// TIA Portal V20 export
FUNCTION_BLOCK "Main_Safety_RTG1"   // FB1, F_LAD
{ S7_Optimized_Access := 'TRUE' }
   VAR
      ESTOP1 : ESTOP1;
   END_VAR
BEGIN

REGION Network 1: Estops on electrical cabins
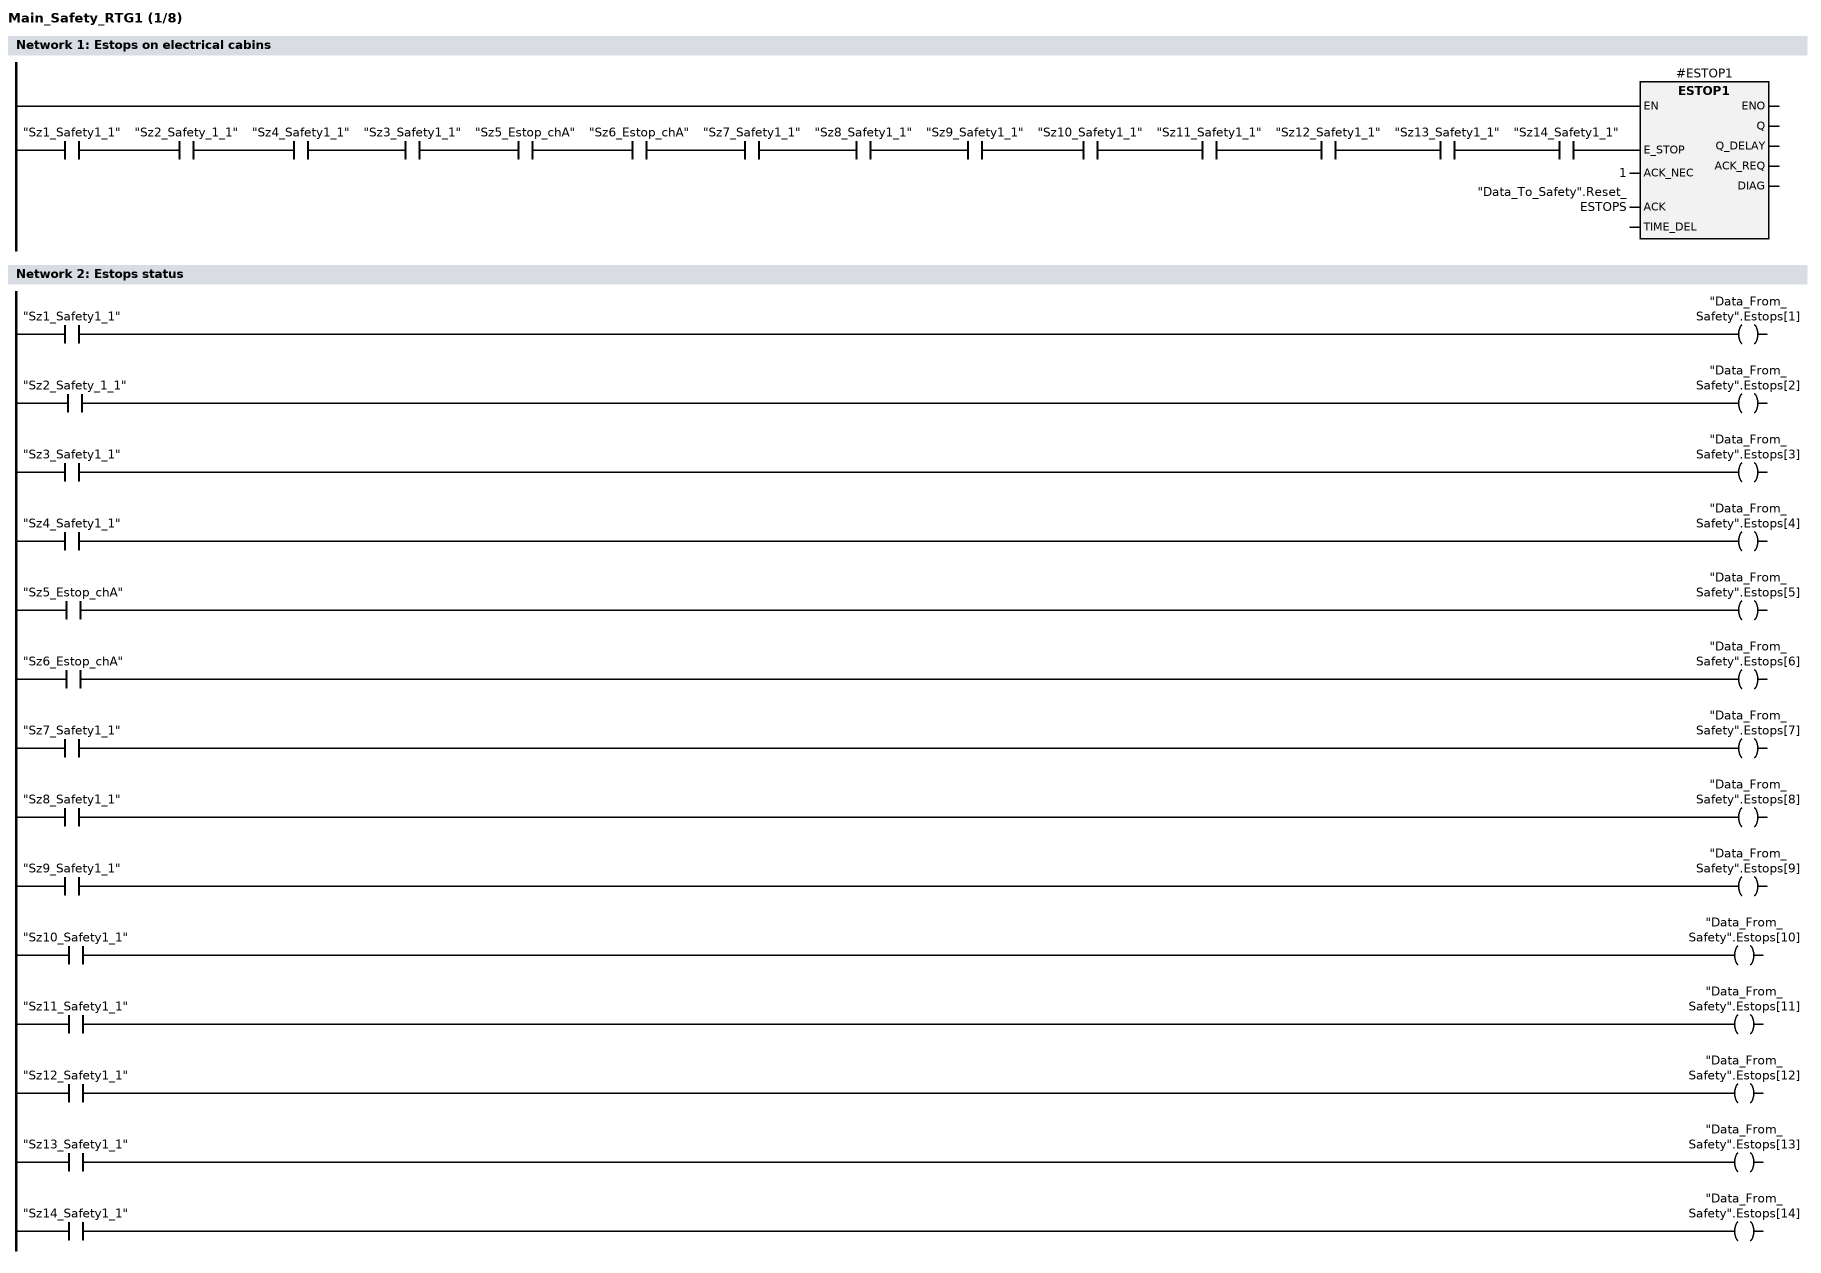
   RUNG wire#powerrail
      #ESTOP1.ESTOP1(E_STOP := wire#w1, ACK_NEC := 1, ACK := "Data_To_Safety".Reset_ESTOPS, TIME_DEL :=, Q =>, Q_DELAY =>, ACK_REQ =>, DIAG =>)
   END_RUNG
   RUNG wire#powerrail
      Contact( "Sz1_Safety1_1" )
      Contact( "Sz2_Safety_1_1" )
      Contact( "Sz4_Safety1_1" )
      Contact( "Sz3_Safety1_1" )
      Contact( "Sz5_Estop_chA" )
      Contact( "Sz6_Estop_chA" )
      Contact( "Sz7_Safety1_1" )
      Contact( "Sz8_Safety1_1" )
      Contact( "Sz9_Safety1_1" )
      Contact( "Sz10_Safety1_1" )
      Contact( "Sz11_Safety1_1" )
      Contact( "Sz12_Safety1_1" )
      Contact( "Sz13_Safety1_1" )
      Contact( "Sz14_Safety1_1" )
   END_RUNG wire#w1
   // the same network as SCL:
   #ESTOP1(E_STOP := "Sz1_Safety1_1" AND "Sz2_Safety_1_1" AND "Sz4_Safety1_1" AND "Sz3_Safety1_1" AND "Sz5_Estop_chA" AND "Sz6_Estop_chA" AND "Sz7_Safety1_1" AND "Sz8_Safety1_1" AND "Sz9_Safety1_1" AND "Sz10_Safety1_1" AND "Sz11_Safety1_1" AND "Sz12_Safety1_1" AND "Sz13_Safety1_1" AND "Sz14_Safety1_1",   // ESTOP1
           ACK_NEC := 1,
           ACK := "Data_To_Safety".Reset_ESTOPS);
END_REGION

REGION Network 2: Estops status
   RUNG wire#powerrail
      Contact( "Sz1_Safety1_1" )
      Coil( "Data_From_Safety".Estops[1] )
   END_RUNG
   RUNG wire#powerrail
      Contact( "Sz2_Safety_1_1" )
      Coil( "Data_From_Safety".Estops[2] )
   END_RUNG
   RUNG wire#powerrail
      Contact( "Sz3_Safety1_1" )
      Coil( "Data_From_Safety".Estops[3] )
   END_RUNG
   RUNG wire#powerrail
      Contact( "Sz4_Safety1_1" )
      Coil( "Data_From_Safety".Estops[4] )
   END_RUNG
   RUNG wire#powerrail
      Contact( "Sz5_Estop_chA" )
      Coil( "Data_From_Safety".Estops[5] )
   END_RUNG
   RUNG wire#powerrail
      Contact( "Sz6_Estop_chA" )
      Coil( "Data_From_Safety".Estops[6] )
   END_RUNG
   RUNG wire#powerrail
      Contact( "Sz7_Safety1_1" )
      Coil( "Data_From_Safety".Estops[7] )
   END_RUNG
   RUNG wire#powerrail
      Contact( "Sz8_Safety1_1" )
      Coil( "Data_From_Safety".Estops[8] )
   END_RUNG
   RUNG wire#powerrail
      Contact( "Sz9_Safety1_1" )
      Coil( "Data_From_Safety".Estops[9] )
   END_RUNG
   RUNG wire#powerrail
      Contact( "Sz10_Safety1_1" )
      Coil( "Data_From_Safety".Estops[10] )
   END_RUNG
   RUNG wire#powerrail
      Contact( "Sz11_Safety1_1" )
      Coil( "Data_From_Safety".Estops[11] )
   END_RUNG
   RUNG wire#powerrail
      Contact( "Sz12_Safety1_1" )
      Coil( "Data_From_Safety".Estops[12] )
   END_RUNG
   RUNG wire#powerrail
      Contact( "Sz13_Safety1_1" )
      Coil( "Data_From_Safety".Estops[13] )
   END_RUNG
   RUNG wire#powerrail
      Contact( "Sz14_Safety1_1" )
      Coil( "Data_From_Safety".Estops[14] )
   END_RUNG
   // the same network as SCL:
   "Data_From_Safety".Estops[1] := "Sz1_Safety1_1";
   "Data_From_Safety".Estops[2] := "Sz2_Safety_1_1";
   "Data_From_Safety".Estops[3] := "Sz3_Safety1_1";
   "Data_From_Safety".Estops[4] := "Sz4_Safety1_1";
   "Data_From_Safety".Estops[5] := "Sz5_Estop_chA";
   "Data_From_Safety".Estops[6] := "Sz6_Estop_chA";
   "Data_From_Safety".Estops[7] := "Sz7_Safety1_1";
   "Data_From_Safety".Estops[8] := "Sz8_Safety1_1";
   "Data_From_Safety".Estops[9] := "Sz9_Safety1_1";
   "Data_From_Safety".Estops[10] := "Sz10_Safety1_1";
   "Data_From_Safety".Estops[11] := "Sz11_Safety1_1";
   "Data_From_Safety".Estops[12] := "Sz12_Safety1_1";
   "Data_From_Safety".Estops[13] := "Sz13_Safety1_1";
   "Data_From_Safety".Estops[14] := "Sz14_Safety1_1";
END_REGION

REGION Network 3: Bumpers SS1_R1
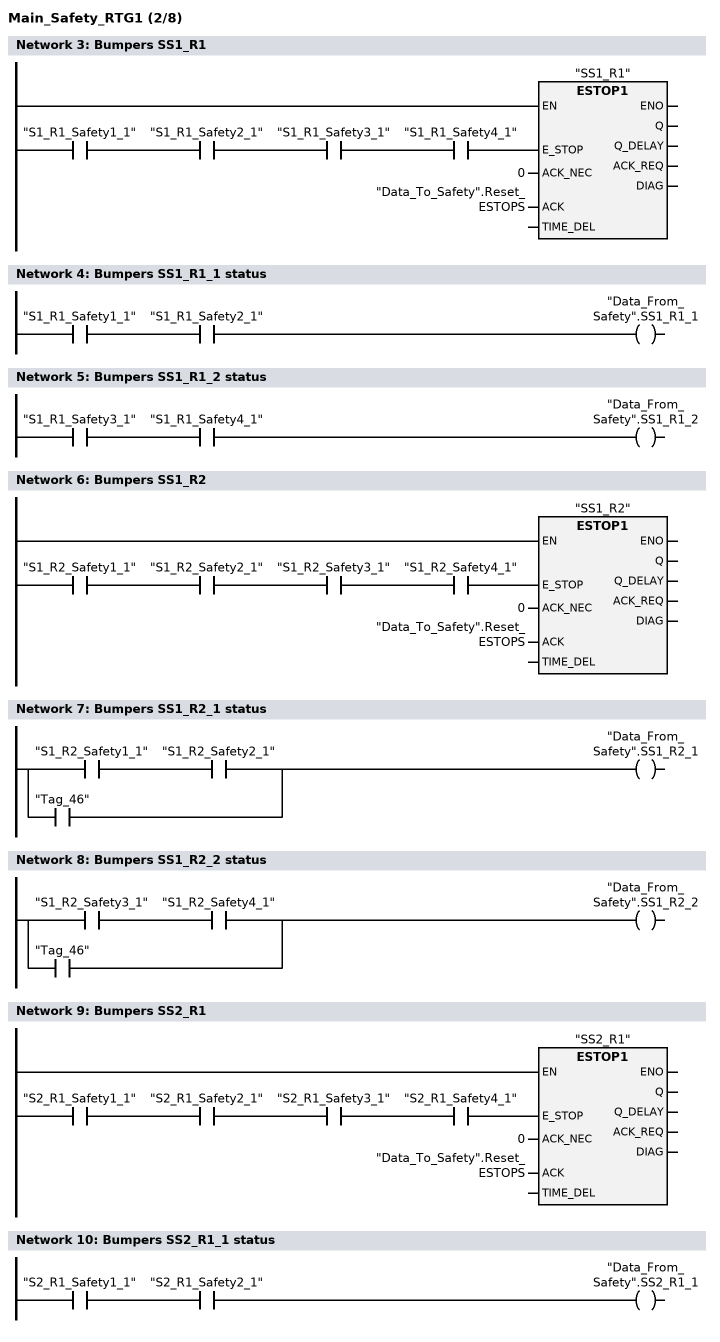
   RUNG wire#powerrail
      "SS1_R1".ESTOP1(E_STOP := wire#w1, ACK_NEC := 0, ACK := "Data_To_Safety".Reset_ESTOPS, TIME_DEL :=, Q =>, Q_DELAY =>, ACK_REQ =>, DIAG =>)
   END_RUNG
   RUNG wire#powerrail
      Contact( "S1_R1_Safety1_1" )
      Contact( "S1_R1_Safety2_1" )
      Contact( "S1_R1_Safety3_1" )
      Contact( "S1_R1_Safety4_1" )
   END_RUNG wire#w1
   // the same network as SCL:
   "SS1_R1"(E_STOP := "S1_R1_Safety1_1" AND "S1_R1_Safety2_1" AND "S1_R1_Safety3_1" AND "S1_R1_Safety4_1",   // ESTOP1
            ACK_NEC := 0,
            ACK := "Data_To_Safety".Reset_ESTOPS);
END_REGION

REGION Network 4: Bumpers SS1_R1_1 status
   RUNG wire#powerrail
      Contact( "S1_R1_Safety1_1" )
      Contact( "S1_R1_Safety2_1" )
      Coil( "Data_From_Safety".SS1_R1_1 )
   END_RUNG
   // the same network as SCL:
   "Data_From_Safety".SS1_R1_1 := "S1_R1_Safety1_1" AND "S1_R1_Safety2_1";
END_REGION

REGION Network 5: Bumpers SS1_R1_2 status
   RUNG wire#powerrail
      Contact( "S1_R1_Safety3_1" )
      Contact( "S1_R1_Safety4_1" )
      Coil( "Data_From_Safety".SS1_R1_2 )
   END_RUNG
   // the same network as SCL:
   "Data_From_Safety".SS1_R1_2 := "S1_R1_Safety3_1" AND "S1_R1_Safety4_1";
END_REGION

REGION Network 6: Bumpers SS1_R2
   RUNG wire#powerrail
      "SS1_R2".ESTOP1(E_STOP := wire#w1, ACK_NEC := 0, ACK := "Data_To_Safety".Reset_ESTOPS, TIME_DEL :=, Q =>, Q_DELAY =>, ACK_REQ =>, DIAG =>)
   END_RUNG
   RUNG wire#powerrail
      Contact( "S1_R2_Safety1_1" )
      Contact( "S1_R2_Safety2_1" )
      Contact( "S1_R2_Safety3_1" )
      Contact( "S1_R2_Safety4_1" )
   END_RUNG wire#w1
   // the same network as SCL:
   "SS1_R2"(E_STOP := "S1_R2_Safety1_1" AND "S1_R2_Safety2_1" AND "S1_R2_Safety3_1" AND "S1_R2_Safety4_1",   // ESTOP1
            ACK_NEC := 0,
            ACK := "Data_To_Safety".Reset_ESTOPS);
END_REGION

REGION Network 7: Bumpers SS1_R2_1 status
   RUNG wire#powerrail
      Contact( "S1_R2_Safety1_1" )
      Contact( "S1_R2_Safety2_1" )
      wire#w1
      Coil( "Data_From_Safety".SS1_R2_1 )
   END_RUNG
   RUNG wire#powerrail
      Contact( "Tag_46" )
   END_RUNG wire#w1
   // the same network as SCL:
   "Data_From_Safety".SS1_R2_1 := ("S1_R2_Safety1_1" AND "S1_R2_Safety2_1") OR "Tag_46";
END_REGION

REGION Network 8: Bumpers SS1_R2_2 status
   RUNG wire#powerrail
      Contact( "S1_R2_Safety3_1" )
      Contact( "S1_R2_Safety4_1" )
      wire#w1
      Coil( "Data_From_Safety".SS1_R2_2 )
   END_RUNG
   RUNG wire#powerrail
      Contact( "Tag_46" )
   END_RUNG wire#w1
   // the same network as SCL:
   "Data_From_Safety".SS1_R2_2 := ("S1_R2_Safety3_1" AND "S1_R2_Safety4_1") OR "Tag_46";
END_REGION

REGION Network 9: Bumpers SS2_R1
   RUNG wire#powerrail
      "SS2_R1".ESTOP1(E_STOP := wire#w1, ACK_NEC := 0, ACK := "Data_To_Safety".Reset_ESTOPS, TIME_DEL :=, Q =>, Q_DELAY =>, ACK_REQ =>, DIAG =>)
   END_RUNG
   RUNG wire#powerrail
      Contact( "S2_R1_Safety1_1" )
      Contact( "S2_R1_Safety2_1" )
      Contact( "S2_R1_Safety3_1" )
      Contact( "S2_R1_Safety4_1" )
   END_RUNG wire#w1
   // the same network as SCL:
   "SS2_R1"(E_STOP := "S2_R1_Safety1_1" AND "S2_R1_Safety2_1" AND "S2_R1_Safety3_1" AND "S2_R1_Safety4_1",   // ESTOP1
            ACK_NEC := 0,
            ACK := "Data_To_Safety".Reset_ESTOPS);
END_REGION

REGION Network 10: Bumpers SS2_R1_1 status
   RUNG wire#powerrail
      Contact( "S2_R1_Safety1_1" )
      Contact( "S2_R1_Safety2_1" )
      Coil( "Data_From_Safety".SS2_R1_1 )
   END_RUNG
   // the same network as SCL:
   "Data_From_Safety".SS2_R1_1 := "S2_R1_Safety1_1" AND "S2_R1_Safety2_1";
END_REGION

REGION Network 11: Bumpers SS2_R1_2 status
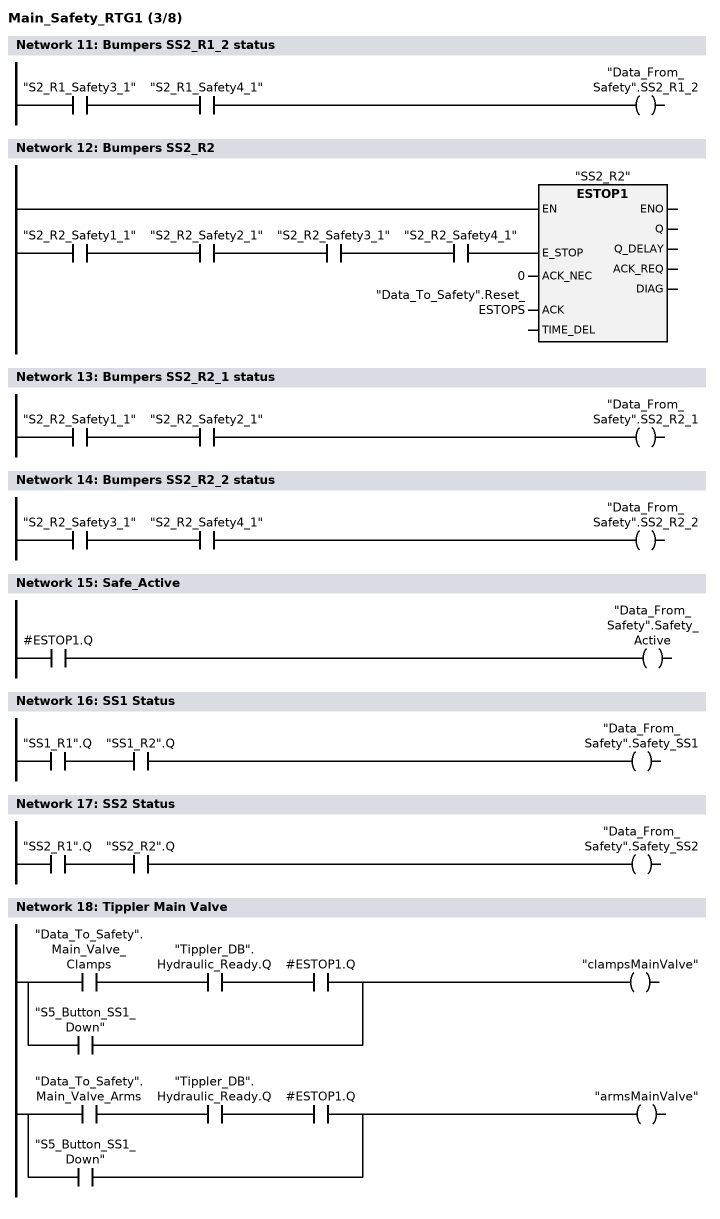
   RUNG wire#powerrail
      Contact( "S2_R1_Safety3_1" )
      Contact( "S2_R1_Safety4_1" )
      Coil( "Data_From_Safety".SS2_R1_2 )
   END_RUNG
   // the same network as SCL:
   "Data_From_Safety".SS2_R1_2 := "S2_R1_Safety3_1" AND "S2_R1_Safety4_1";
END_REGION

REGION Network 12: Bumpers SS2_R2
   RUNG wire#powerrail
      "SS2_R2".ESTOP1(E_STOP := wire#w1, ACK_NEC := 0, ACK := "Data_To_Safety".Reset_ESTOPS, TIME_DEL :=, Q =>, Q_DELAY =>, ACK_REQ =>, DIAG =>)
   END_RUNG
   RUNG wire#powerrail
      Contact( "S2_R2_Safety1_1" )
      Contact( "S2_R2_Safety2_1" )
      Contact( "S2_R2_Safety3_1" )
      Contact( "S2_R2_Safety4_1" )
   END_RUNG wire#w1
   // the same network as SCL:
   "SS2_R2"(E_STOP := "S2_R2_Safety1_1" AND "S2_R2_Safety2_1" AND "S2_R2_Safety3_1" AND "S2_R2_Safety4_1",   // ESTOP1
            ACK_NEC := 0,
            ACK := "Data_To_Safety".Reset_ESTOPS);
END_REGION

REGION Network 13: Bumpers SS2_R2_1 status
   RUNG wire#powerrail
      Contact( "S2_R2_Safety1_1" )
      Contact( "S2_R2_Safety2_1" )
      Coil( "Data_From_Safety".SS2_R2_1 )
   END_RUNG
   // the same network as SCL:
   "Data_From_Safety".SS2_R2_1 := "S2_R2_Safety1_1" AND "S2_R2_Safety2_1";
END_REGION

REGION Network 14: Bumpers SS2_R2_2 status
   RUNG wire#powerrail
      Contact( "S2_R2_Safety3_1" )
      Contact( "S2_R2_Safety4_1" )
      Coil( "Data_From_Safety".SS2_R2_2 )
   END_RUNG
   // the same network as SCL:
   "Data_From_Safety".SS2_R2_2 := "S2_R2_Safety3_1" AND "S2_R2_Safety4_1";
END_REGION

REGION Network 15: Safe_Active
   RUNG wire#powerrail
      Contact( #ESTOP1.Q )
      Coil( "Data_From_Safety".Safety_Active )
   END_RUNG
   // the same network as SCL:
   "Data_From_Safety".Safety_Active := #ESTOP1.Q;
END_REGION

REGION Network 16: SS1 Status
   RUNG wire#powerrail
      Contact( "SS1_R1".Q )
      Contact( "SS1_R2".Q )
      Coil( "Data_From_Safety".Safety_SS1 )
   END_RUNG
   // the same network as SCL:
   "Data_From_Safety".Safety_SS1 := "SS1_R1".Q AND "SS1_R2".Q;
END_REGION

REGION Network 17: SS2 Status
   RUNG wire#powerrail
      Contact( "SS2_R1".Q )
      Contact( "SS2_R2".Q )
      Coil( "Data_From_Safety".Safety_SS2 )
   END_RUNG
   // the same network as SCL:
   "Data_From_Safety".Safety_SS2 := "SS2_R1".Q AND "SS2_R2".Q;
END_REGION

REGION Network 18: Tippler Main Valve
   RUNG wire#powerrail
      Contact( "Data_To_Safety".Main_Valve_Clamps )
      Contact( "Tippler_DB".Hydraulic_Ready.Q )
      Contact( #ESTOP1.Q )
      wire#w1
      Coil( "clampsMainValve" )
   END_RUNG
   RUNG wire#powerrail
      Contact( "S5_Button_SS1_Down" )
   END_RUNG wire#w1
   RUNG wire#powerrail
      Contact( "Data_To_Safety".Main_Valve_Arms )
      Contact( "Tippler_DB".Hydraulic_Ready.Q )
      Contact( #ESTOP1.Q )
      wire#w2
      Coil( "armsMainValve" )
   END_RUNG
   RUNG wire#powerrail
      Contact( "S5_Button_SS1_Down" )
   END_RUNG wire#w2
   // the same network as SCL:
   "clampsMainValve" := ("Data_To_Safety".Main_Valve_Clamps AND "Tippler_DB".Hydraulic_Ready.Q AND #ESTOP1.Q) OR "S5_Button_SS1_Down";
   "armsMainValve" := ("Data_To_Safety".Main_Valve_Arms AND "Tippler_DB".Hydraulic_Ready.Q AND #ESTOP1.Q) OR "S5_Button_SS1_Down";
END_REGION

REGION Network 19: S0_R1, S0_R2
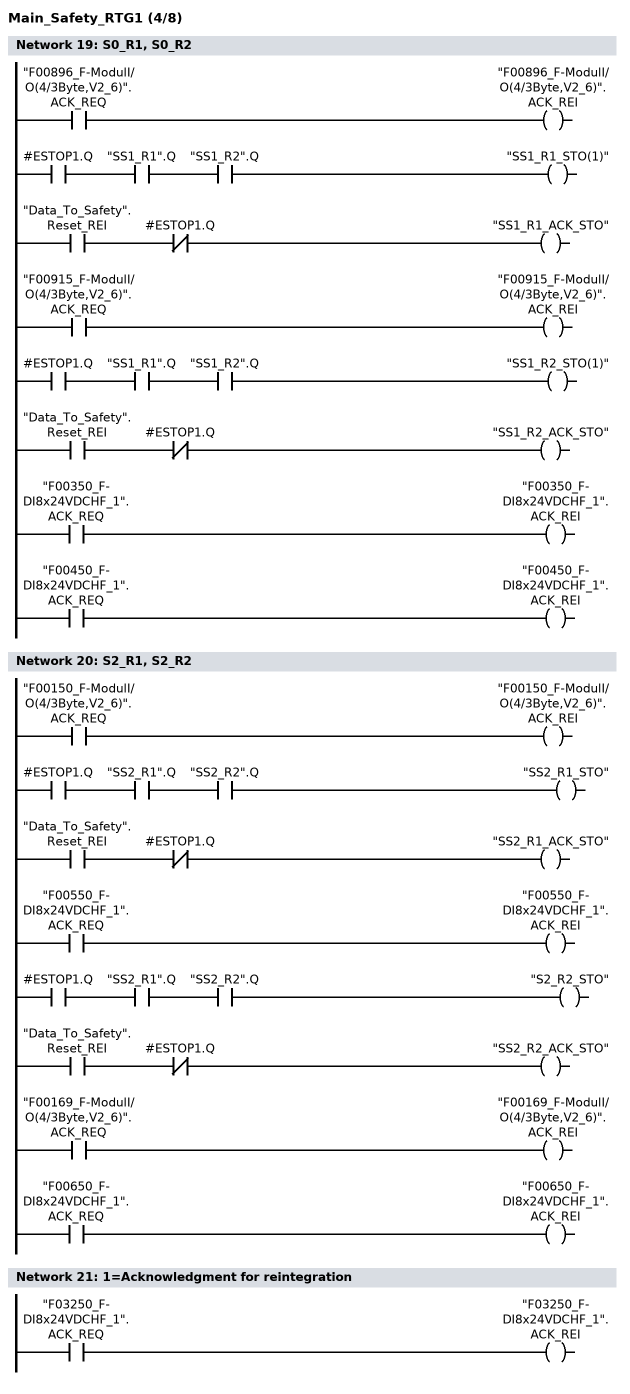
   RUNG wire#powerrail
      Contact( "F00896_F-ModulI/O(4/3Byte,V2_6)".ACK_REQ )
      Coil( "F00896_F-ModulI/O(4/3Byte,V2_6)".ACK_REI )
   END_RUNG
   RUNG wire#powerrail
      Contact( #ESTOP1.Q )
      Contact( "SS1_R1".Q )
      Contact( "SS1_R2".Q )
      Coil( "SS1_R1_STO(1)" )
   END_RUNG
   RUNG wire#powerrail
      Contact( "Data_To_Safety".Reset_REI )
      I_Contact( #ESTOP1.Q )
      Coil( "SS1_R1_ACK_STO" )
   END_RUNG
   RUNG wire#powerrail
      Contact( "F00915_F-ModulI/O(4/3Byte,V2_6)".ACK_REQ )
      Coil( "F00915_F-ModulI/O(4/3Byte,V2_6)".ACK_REI )
   END_RUNG
   RUNG wire#powerrail
      Contact( #ESTOP1.Q )
      Contact( "SS1_R1".Q )
      Contact( "SS1_R2".Q )
      Coil( "SS1_R2_STO(1)" )
   END_RUNG
   RUNG wire#powerrail
      Contact( "Data_To_Safety".Reset_REI )
      I_Contact( #ESTOP1.Q )
      Coil( "SS1_R2_ACK_STO" )
   END_RUNG
   RUNG wire#powerrail
      Contact( "F00350_F-DI8x24VDCHF_1".ACK_REQ )
      Coil( "F00350_F-DI8x24VDCHF_1".ACK_REI )
   END_RUNG
   RUNG wire#powerrail
      Contact( "F00450_F-DI8x24VDCHF_1".ACK_REQ )
      Coil( "F00450_F-DI8x24VDCHF_1".ACK_REI )
   END_RUNG
   // the same network as SCL:
   "F00896_F-ModulI/O(4/3Byte,V2_6)".ACK_REI := "F00896_F-ModulI/O(4/3Byte,V2_6)".ACK_REQ;
   "SS1_R1_STO(1)" := #ESTOP1.Q AND "SS1_R1".Q AND "SS1_R2".Q;
   "SS1_R1_ACK_STO" := "Data_To_Safety".Reset_REI AND NOT #ESTOP1.Q;
   "F00915_F-ModulI/O(4/3Byte,V2_6)".ACK_REI := "F00915_F-ModulI/O(4/3Byte,V2_6)".ACK_REQ;
   "SS1_R2_STO(1)" := #ESTOP1.Q AND "SS1_R1".Q AND "SS1_R2".Q;
   "SS1_R2_ACK_STO" := "Data_To_Safety".Reset_REI AND NOT #ESTOP1.Q;
   "F00350_F-DI8x24VDCHF_1".ACK_REI := "F00350_F-DI8x24VDCHF_1".ACK_REQ;
   "F00450_F-DI8x24VDCHF_1".ACK_REI := "F00450_F-DI8x24VDCHF_1".ACK_REQ;
END_REGION

REGION Network 20: S2_R1, S2_R2
   RUNG wire#powerrail
      Contact( "F00150_F-ModulI/O(4/3Byte,V2_6)".ACK_REQ )
      Coil( "F00150_F-ModulI/O(4/3Byte,V2_6)".ACK_REI )
   END_RUNG
   RUNG wire#powerrail
      Contact( #ESTOP1.Q )
      Contact( "SS2_R1".Q )
      Contact( "SS2_R2".Q )
      Coil( "SS2_R1_STO" )
   END_RUNG
   RUNG wire#powerrail
      Contact( "Data_To_Safety".Reset_REI )
      I_Contact( #ESTOP1.Q )
      Coil( "SS2_R1_ACK_STO" )
   END_RUNG
   RUNG wire#powerrail
      Contact( "F00550_F-DI8x24VDCHF_1".ACK_REQ )
      Coil( "F00550_F-DI8x24VDCHF_1".ACK_REI )
   END_RUNG
   RUNG wire#powerrail
      Contact( #ESTOP1.Q )
      Contact( "SS2_R1".Q )
      Contact( "SS2_R2".Q )
      Coil( "S2_R2_STO" )
   END_RUNG
   RUNG wire#powerrail
      Contact( "Data_To_Safety".Reset_REI )
      I_Contact( #ESTOP1.Q )
      Coil( "SS2_R2_ACK_STO" )
   END_RUNG
   RUNG wire#powerrail
      Contact( "F00169_F-ModulI/O(4/3Byte,V2_6)".ACK_REQ )
      Coil( "F00169_F-ModulI/O(4/3Byte,V2_6)".ACK_REI )
   END_RUNG
   RUNG wire#powerrail
      Contact( "F00650_F-DI8x24VDCHF_1".ACK_REQ )
      Coil( "F00650_F-DI8x24VDCHF_1".ACK_REI )
   END_RUNG
   // the same network as SCL:
   "F00150_F-ModulI/O(4/3Byte,V2_6)".ACK_REI := "F00150_F-ModulI/O(4/3Byte,V2_6)".ACK_REQ;
   "SS2_R1_STO" := #ESTOP1.Q AND "SS2_R1".Q AND "SS2_R2".Q;
   "SS2_R1_ACK_STO" := "Data_To_Safety".Reset_REI AND NOT #ESTOP1.Q;
   "F00550_F-DI8x24VDCHF_1".ACK_REI := "F00550_F-DI8x24VDCHF_1".ACK_REQ;
   "S2_R2_STO" := #ESTOP1.Q AND "SS2_R1".Q AND "SS2_R2".Q;
   "SS2_R2_ACK_STO" := "Data_To_Safety".Reset_REI AND NOT #ESTOP1.Q;
   "F00169_F-ModulI/O(4/3Byte,V2_6)".ACK_REI := "F00169_F-ModulI/O(4/3Byte,V2_6)".ACK_REQ;
   "F00650_F-DI8x24VDCHF_1".ACK_REI := "F00650_F-DI8x24VDCHF_1".ACK_REQ;
END_REGION

REGION Network 21: 1=Acknowledgment for reintegration
   RUNG wire#powerrail
      Contact( "F03250_F-DI8x24VDCHF_1".ACK_REQ )
      Coil( "F03250_F-DI8x24VDCHF_1".ACK_REI )
   END_RUNG
   // the same network as SCL:
   "F03250_F-DI8x24VDCHF_1".ACK_REI := "F03250_F-DI8x24VDCHF_1".ACK_REQ;
END_REGION

REGION Network 22: ROW 1
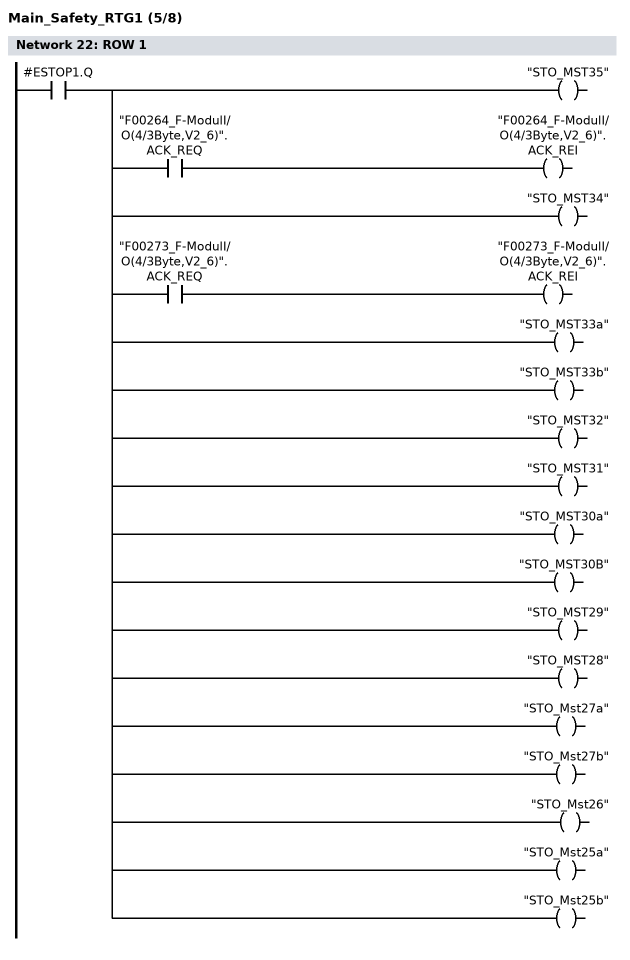
   RUNG wire#powerrail
      Contact( #ESTOP1.Q )
      wire#w1
      Coil( "STO_MST35" )
   END_RUNG
   RUNG wire#w1
      Contact( "F00264_F-ModulI/O(4/3Byte,V2_6)".ACK_REQ )
      Coil( "F00264_F-ModulI/O(4/3Byte,V2_6)".ACK_REI )
   END_RUNG
   RUNG wire#w1
      Coil( "STO_MST34" )
   END_RUNG
   RUNG wire#w1
      Contact( "F00273_F-ModulI/O(4/3Byte,V2_6)".ACK_REQ )
      Coil( "F00273_F-ModulI/O(4/3Byte,V2_6)".ACK_REI )
   END_RUNG
   RUNG wire#w1
      Coil( "STO_MST33a" )
   END_RUNG
   RUNG wire#w1
      Coil( "STO_MST33b" )
   END_RUNG
   RUNG wire#w1
      Coil( "STO_MST32" )
   END_RUNG
   RUNG wire#w1
      Coil( "STO_MST31" )
   END_RUNG
   RUNG wire#w1
      Coil( "STO_MST30a" )
   END_RUNG
   RUNG wire#w1
      Coil( "STO_MST30B" )
   END_RUNG
   RUNG wire#w1
      Coil( "STO_MST29" )
   END_RUNG
   RUNG wire#w1
      Coil( "STO_MST28" )
   END_RUNG
   RUNG wire#w1
      Coil( "STO_Mst27a" )
   END_RUNG
   RUNG wire#w1
      Coil( "STO_Mst27b" )
   END_RUNG
   RUNG wire#w1
      Coil( "STO_Mst26" )
   END_RUNG
   RUNG wire#w1
      Coil( "STO_Mst25a" )
   END_RUNG
   RUNG wire#w1
      Coil( "STO_Mst25b" )
   END_RUNG
   // the same network as SCL:
   "STO_MST35" := #ESTOP1.Q;
   "F00264_F-ModulI/O(4/3Byte,V2_6)".ACK_REI := #ESTOP1.Q AND "F00264_F-ModulI/O(4/3Byte,V2_6)".ACK_REQ;
   "STO_MST34" := #ESTOP1.Q;
   "F00273_F-ModulI/O(4/3Byte,V2_6)".ACK_REI := #ESTOP1.Q AND "F00273_F-ModulI/O(4/3Byte,V2_6)".ACK_REQ;
   "STO_MST33a" := #ESTOP1.Q;
   "STO_MST33b" := #ESTOP1.Q;
   "STO_MST32" := #ESTOP1.Q;
   "STO_MST31" := #ESTOP1.Q;
   "STO_MST30a" := #ESTOP1.Q;
   "STO_MST30B" := #ESTOP1.Q;
   "STO_MST29" := #ESTOP1.Q;
   "STO_MST28" := #ESTOP1.Q;
   "STO_Mst27a" := #ESTOP1.Q;
   "STO_Mst27b" := #ESTOP1.Q;
   "STO_Mst26" := #ESTOP1.Q;
   "STO_Mst25a" := #ESTOP1.Q;
   "STO_Mst25b" := #ESTOP1.Q;
END_REGION

REGION Network 23: ROW 2
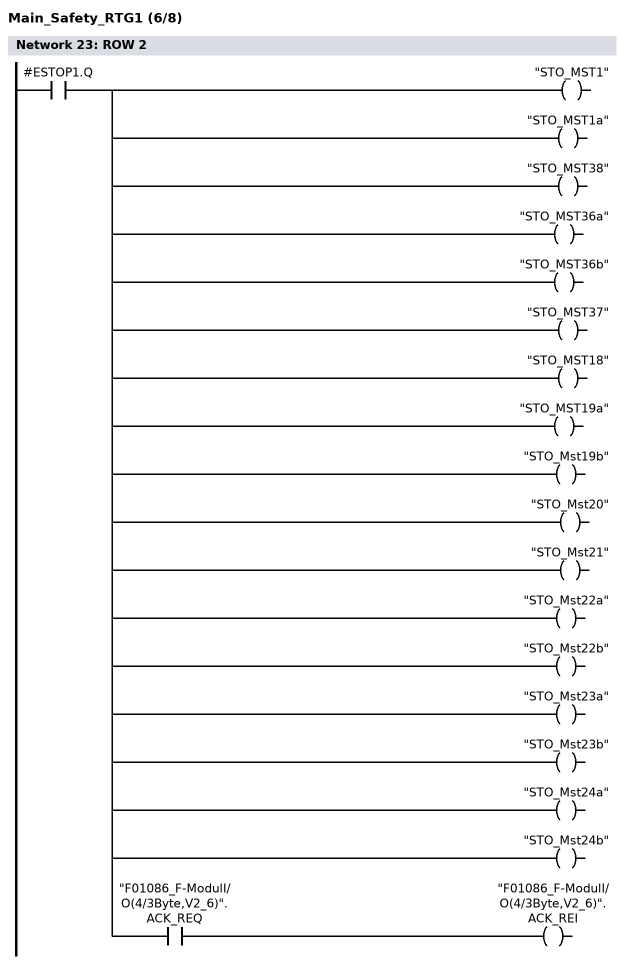
   RUNG wire#powerrail
      Contact( #ESTOP1.Q )
      wire#w1
      Coil( "STO_MST1" )
   END_RUNG
   RUNG wire#w1
      Coil( "STO_MST1a" )
   END_RUNG
   RUNG wire#w1
      Coil( "STO_MST38" )
   END_RUNG
   RUNG wire#w1
      Coil( "STO_MST36a" )
   END_RUNG
   RUNG wire#w1
      Coil( "STO_MST36b" )
   END_RUNG
   RUNG wire#w1
      Coil( "STO_MST37" )
   END_RUNG
   RUNG wire#w1
      Coil( "STO_MST18" )
   END_RUNG
   RUNG wire#w1
      Coil( "STO_MST19a" )
   END_RUNG
   RUNG wire#w1
      Coil( "STO_Mst19b" )
   END_RUNG
   RUNG wire#w1
      Coil( "STO_Mst20" )
   END_RUNG
   RUNG wire#w1
      Coil( "STO_Mst21" )
   END_RUNG
   RUNG wire#w1
      Coil( "STO_Mst22a" )
   END_RUNG
   RUNG wire#w1
      Coil( "STO_Mst22b" )
   END_RUNG
   RUNG wire#w1
      Coil( "STO_Mst23a" )
   END_RUNG
   RUNG wire#w1
      Coil( "STO_Mst23b" )
   END_RUNG
   RUNG wire#w1
      Coil( "STO_Mst24a" )
   END_RUNG
   RUNG wire#w1
      Coil( "STO_Mst24b" )
   END_RUNG
   RUNG wire#w1
      Contact( "F01086_F-ModulI/O(4/3Byte,V2_6)".ACK_REQ )
      Coil( "F01086_F-ModulI/O(4/3Byte,V2_6)".ACK_REI )
   END_RUNG
   // the same network as SCL:
   "STO_MST1" := #ESTOP1.Q;
   "STO_MST1a" := #ESTOP1.Q;
   "STO_MST38" := #ESTOP1.Q;
   "STO_MST36a" := #ESTOP1.Q;
   "STO_MST36b" := #ESTOP1.Q;
   "STO_MST37" := #ESTOP1.Q;
   "STO_MST18" := #ESTOP1.Q;
   "STO_MST19a" := #ESTOP1.Q;
   "STO_Mst19b" := #ESTOP1.Q;
   "STO_Mst20" := #ESTOP1.Q;
   "STO_Mst21" := #ESTOP1.Q;
   "STO_Mst22a" := #ESTOP1.Q;
   "STO_Mst22b" := #ESTOP1.Q;
   "STO_Mst23a" := #ESTOP1.Q;
   "STO_Mst23b" := #ESTOP1.Q;
   "STO_Mst24a" := #ESTOP1.Q;
   "STO_Mst24b" := #ESTOP1.Q;
   "F01086_F-ModulI/O(4/3Byte,V2_6)".ACK_REI := #ESTOP1.Q AND "F01086_F-ModulI/O(4/3Byte,V2_6)".ACK_REQ;
END_REGION

REGION Network 24: ROW 4
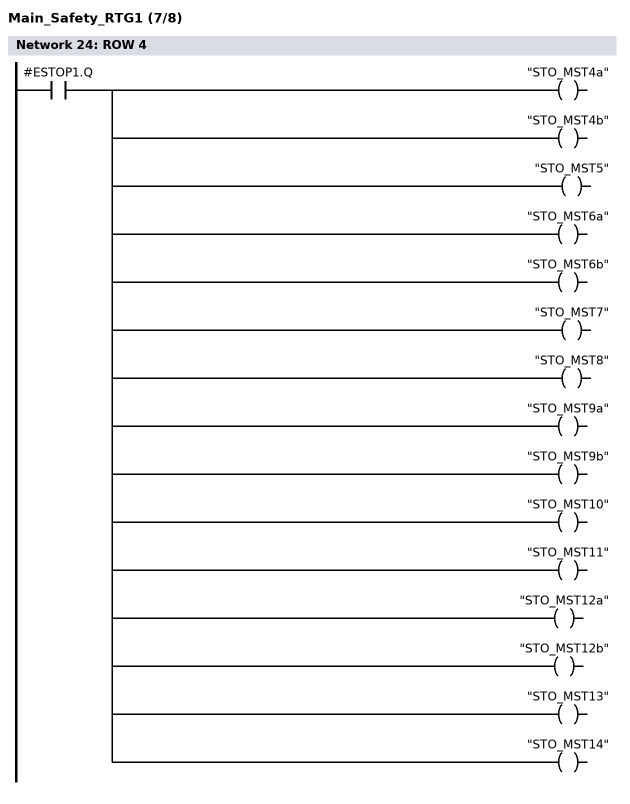
   RUNG wire#powerrail
      Contact( #ESTOP1.Q )
      wire#w1
      Coil( "STO_MST4a" )
   END_RUNG
   RUNG wire#w1
      Coil( "STO_MST4b" )
   END_RUNG
   RUNG wire#w1
      Coil( "STO_MST5" )
   END_RUNG
   RUNG wire#w1
      Coil( "STO_MST6a" )
   END_RUNG
   RUNG wire#w1
      Coil( "STO_MST6b" )
   END_RUNG
   RUNG wire#w1
      Coil( "STO_MST7" )
   END_RUNG
   RUNG wire#w1
      Coil( "STO_MST8" )
   END_RUNG
   RUNG wire#w1
      Coil( "STO_MST9a" )
   END_RUNG
   RUNG wire#w1
      Coil( "STO_MST9b" )
   END_RUNG
   RUNG wire#w1
      Coil( "STO_MST10" )
   END_RUNG
   RUNG wire#w1
      Coil( "STO_MST11" )
   END_RUNG
   RUNG wire#w1
      Coil( "STO_MST12a" )
   END_RUNG
   RUNG wire#w1
      Coil( "STO_MST12b" )
   END_RUNG
   RUNG wire#w1
      Coil( "STO_MST13" )
   END_RUNG
   RUNG wire#w1
      Coil( "STO_MST14" )
   END_RUNG
   // the same network as SCL:
   "STO_MST4a" := #ESTOP1.Q;
   "STO_MST4b" := #ESTOP1.Q;
   "STO_MST5" := #ESTOP1.Q;
   "STO_MST6a" := #ESTOP1.Q;
   "STO_MST6b" := #ESTOP1.Q;
   "STO_MST7" := #ESTOP1.Q;
   "STO_MST8" := #ESTOP1.Q;
   "STO_MST9a" := #ESTOP1.Q;
   "STO_MST9b" := #ESTOP1.Q;
   "STO_MST10" := #ESTOP1.Q;
   "STO_MST11" := #ESTOP1.Q;
   "STO_MST12a" := #ESTOP1.Q;
   "STO_MST12b" := #ESTOP1.Q;
   "STO_MST13" := #ESTOP1.Q;
   "STO_MST14" := #ESTOP1.Q;
END_REGION

REGION Network 25: CS
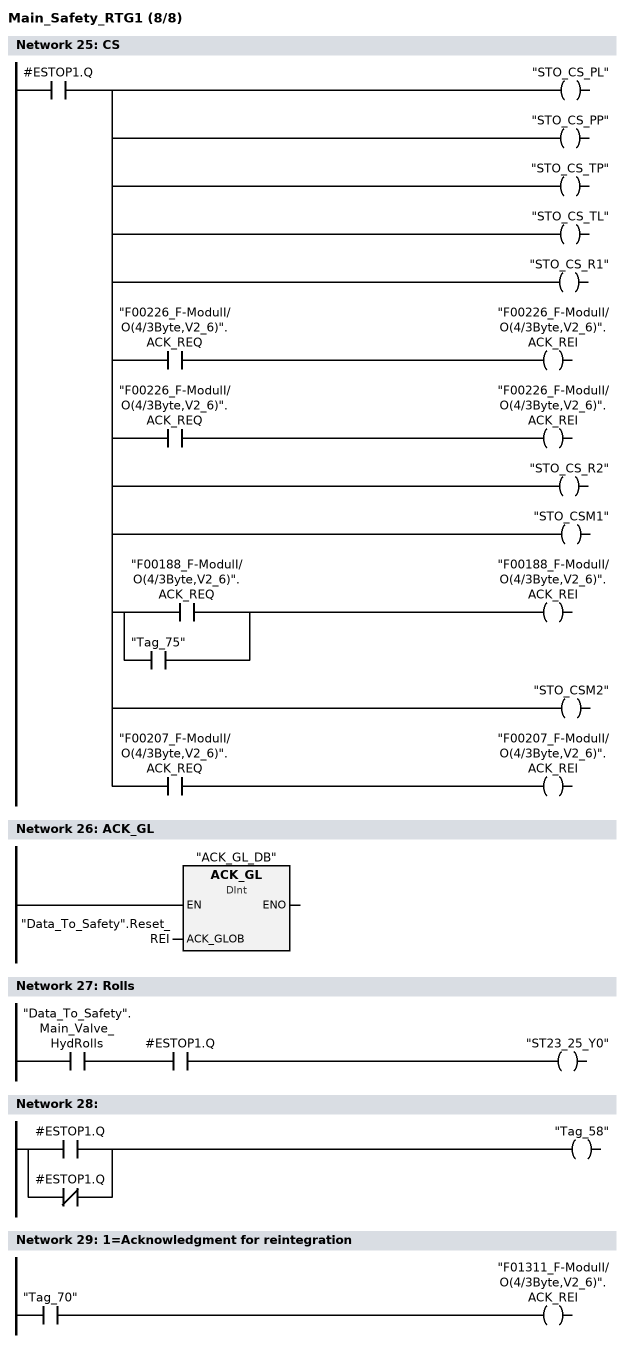
   RUNG wire#powerrail
      Contact( #ESTOP1.Q )
      wire#w1
      Coil( "STO_CS_PL" )
   END_RUNG
   RUNG wire#w1
      Coil( "STO_CS_PP" )
   END_RUNG
   RUNG wire#w1
      Coil( "STO_CS_TP" )
   END_RUNG
   RUNG wire#w1
      Coil( "STO_CS_TL" )
   END_RUNG
   RUNG wire#w1
      Coil( "STO_CS_R1" )
   END_RUNG
   RUNG wire#w1
      Contact( "F00226_F-ModulI/O(4/3Byte,V2_6)".ACK_REQ )
      Coil( "F00226_F-ModulI/O(4/3Byte,V2_6)".ACK_REI )
   END_RUNG
   RUNG wire#w1
      Contact( "F00226_F-ModulI/O(4/3Byte,V2_6)".ACK_REQ )
      Coil( "F00226_F-ModulI/O(4/3Byte,V2_6)".ACK_REI )
   END_RUNG
   RUNG wire#w1
      Coil( "STO_CS_R2" )
   END_RUNG
   RUNG wire#w1
      Coil( "STO_CSM1" )
   END_RUNG
   RUNG wire#w1
      Contact( "F00188_F-ModulI/O(4/3Byte,V2_6)".ACK_REQ )
      wire#w2
      Coil( "F00188_F-ModulI/O(4/3Byte,V2_6)".ACK_REI )
   END_RUNG
   RUNG wire#w1
      Contact( "Tag_75" )
   END_RUNG wire#w2
   RUNG wire#w1
      Coil( "STO_CSM2" )
   END_RUNG
   RUNG wire#w1
      Contact( "F00207_F-ModulI/O(4/3Byte,V2_6)".ACK_REQ )
      Coil( "F00207_F-ModulI/O(4/3Byte,V2_6)".ACK_REI )
   END_RUNG
   // the same network as SCL:
   "STO_CS_PL" := #ESTOP1.Q;
   "STO_CS_PP" := #ESTOP1.Q;
   "STO_CS_TP" := #ESTOP1.Q;
   "STO_CS_TL" := #ESTOP1.Q;
   "STO_CS_R1" := #ESTOP1.Q;
   "F00226_F-ModulI/O(4/3Byte,V2_6)".ACK_REI := #ESTOP1.Q AND "F00226_F-ModulI/O(4/3Byte,V2_6)".ACK_REQ;
   "F00226_F-ModulI/O(4/3Byte,V2_6)".ACK_REI := #ESTOP1.Q AND "F00226_F-ModulI/O(4/3Byte,V2_6)".ACK_REQ;
   "STO_CS_R2" := #ESTOP1.Q;
   "STO_CSM1" := #ESTOP1.Q;
   "F00188_F-ModulI/O(4/3Byte,V2_6)".ACK_REI := #ESTOP1.Q AND ("F00188_F-ModulI/O(4/3Byte,V2_6)".ACK_REQ OR "Tag_75");
   "STO_CSM2" := #ESTOP1.Q;
   "F00207_F-ModulI/O(4/3Byte,V2_6)".ACK_REI := #ESTOP1.Q AND "F00207_F-ModulI/O(4/3Byte,V2_6)".ACK_REQ;
END_REGION

REGION Network 26: ACK_GL
   RUNG wire#powerrail
      { S7_Templates := "codedbool_type := DInt" } "ACK_GL_DB".ACK_GL(ACK_GLOB := "Data_To_Safety".Reset_REI)
   END_RUNG
   // the same network as SCL:
   "ACK_GL_DB"(ACK_GLOB := "Data_To_Safety".Reset_REI);   // ACK_GL
END_REGION

REGION Network 27: Rolls
   RUNG wire#powerrail
      Contact( "Data_To_Safety".Main_Valve_HydRolls )
      Contact( #ESTOP1.Q )
      Coil( "ST23_25_Y0" )
   END_RUNG
   // the same network as SCL:
   "ST23_25_Y0" := "Data_To_Safety".Main_Valve_HydRolls AND #ESTOP1.Q;
END_REGION

REGION Network 28
   RUNG wire#powerrail
      Contact( #ESTOP1.Q )
      wire#w1
      Coil( "Tag_58" )
   END_RUNG
   RUNG wire#powerrail
      I_Contact( #ESTOP1.Q )
   END_RUNG wire#w1
   // the same network as SCL:
   "Tag_58" := #ESTOP1.Q OR NOT #ESTOP1.Q;
END_REGION

REGION Network 29: 1=Acknowledgment for reintegration
   RUNG wire#powerrail
      Contact( "Tag_70" )
      Coil( "F01311_F-ModulI/O(4/3Byte,V2_6)".ACK_REI )
   END_RUNG
   // the same network as SCL:
   "F01311_F-ModulI/O(4/3Byte,V2_6)".ACK_REI := "Tag_70";
END_REGION
END_FUNCTION_BLOCK
